// TwinCAT 3 PLC project PidTests
// ProgramVersion: 3.1.4026.22
// libraries:
//   Tc2_Standard, * (Beckhoff Automation GmbH)
//   Tc2_System, * (Beckhoff Automation GmbH)
//   TcUnit, * (www.tcunit.org)
//   T2Pid_Plc,newest,Tc3 Project
// project tree:
//   / PlcTask.TcTTO
//   POUs/ FB_PidTests.TcPOU, MAIN.TcPOU
// real-time tasks:
//   TASK PlcTask: cycle T#10ms, priority 20, ADS port 350

CONFIGURATION PidTests
    RESOURCE PLC ON TwinCAT3
        TASK PlcTask(INTERVAL := T#10ms, PRIORITY := 20);
        PROGRAM MAIN WITH PlcTask : MAIN;
    END_RESOURCE
END_CONFIGURATION

// ---- POUs/MAIN.TcPOU
PROGRAM MAIN
VAR
    suite : FB_PidTests;
END_VAR

suite();
TcUnit.RUN();

END_PROGRAM

// ---- POUs/FB_PidTests.TcPOU
FUNCTION_BLOCK FB_PidTests EXTENDS TcUnit.FB_TestSuite
VAR
    pid       : T2Pid_Plc.FB_Pid;
    iPid      : T2Pid_Plc.I_Pid;
    output    : LREAL;
    output2   : LREAL;
    integral  : LREAL;
    saturated : BOOL;
    i         : DINT;
END_VAR

PProportionalOnly();
OutputClampsToMax();
OutputClampsToMin();
IntegralAccumulates();
AntiWindupHoldsIntegral();
DerivativeOnMeasurementNoSetpointSpike();
ReverseModeFlipsSign();
ResetClearsIntegral();
SetterRejectsNegativeKp();
IsSaturatedReflectsClampState();
CyclicReachableThroughInterface();

METHOD AntiWindupHoldsIntegral : BOOL
VAR
    integral : LREAL;
    i : DINT;
END_VAR
IF TEST_ORDERED(__POUNAME()) THEN
    pid.Reset();
    pid.Kp := 0.0;
    pid.Ki := 10.0;
    pid.Kd := 0.0;
    pid.Mode := 0;
    pid.OutputMin := -1.0;
    pid.OutputMax := 1.0;
    // Drive into saturation: with Ki=10 and error=1, a single 0.1s tick
    // would produce output 1.0 (at clamp). Twenty more ticks should
    // not grow the integral once saturated.
    FOR i := 1 TO 20 DO
        pid.Update(setpoint := 1.0, measurement := 0.0, deltaT := 0.1);
    END_FOR
    integral := pid.IntegralTerm;
    AssertTrue(Condition := integral <= 0.2,
        Message := 'Anti-windup should hold integral at/near saturation point, not let it grow');
    TEST_FINISHED();
END_IF
END_METHOD

METHOD CyclicReachableThroughInterface : BOOL
VAR
    direct    : LREAL;
    viaIface  : LREAL;
END_VAR
IF TEST_ORDERED(__POUNAME()) THEN
    pid.Reset();
    pid.Kp := 3.0;
    pid.Ki := 0.0;
    pid.Kd := 0.0;
    pid.Mode := 0;
    pid.OutputMin := -100.0;
    pid.OutputMax := 100.0;
    direct := pid.Update(setpoint := 1.0, measurement := 0.0, deltaT := 0.1);

    pid.Reset();
    iPid := pid;  // FB_Pid IMPLEMENTS I_Pid required
    viaIface := iPid.Update(setpoint := 1.0, measurement := 0.0, deltaT := 0.1);

    AssertEquals_LREAL(Expected := direct, Actual := viaIface, Delta := 1E-9,
        Message := 'Same Update inputs through pid and iPid must give the same output');
    TEST_FINISHED();
END_IF
END_METHOD

METHOD DerivativeOnMeasurementNoSetpointSpike : BOOL
VAR
    output : LREAL;
    output2 : LREAL;
END_VAR
IF TEST_ORDERED(__POUNAME()) THEN
    pid.Reset();
    pid.Kp := 0.0;
    pid.Ki := 0.0;
    pid.Kd := 1.0;
    pid.Mode := 0;
    pid.OutputMin := -100.0;
    pid.OutputMax := 100.0;
    // Steady state: setpoint=0, measurement=0.
    pid.Update(setpoint := 0.0, measurement := 0.0, deltaT := 0.1);
    // Step the SETPOINT. With derivative-on-error this would produce
    // a large spike (d_error/dt ~ 100). With derivative-on-measurement
    // the derivative is computed from -dMeasurement/dt, which is 0.
    output := pid.Update(setpoint := 10.0, measurement := 0.0, deltaT := 0.1);
    AssertTrue(Condition := ABS(output) < 1.0,
        Message := 'Derivative-on-measurement: setpoint step must NOT cause D-kick');
    TEST_FINISHED();
END_IF
END_METHOD

METHOD IntegralAccumulates : BOOL
VAR
    integral : LREAL;
    i : DINT;
END_VAR
IF TEST_ORDERED(__POUNAME()) THEN
    pid.Reset();
    pid.Kp := 0.0;
    pid.Ki := 1.0;
    pid.Kd := 0.0;
    pid.Mode := 0;
    pid.OutputMin := -100.0;
    pid.OutputMax := 100.0;
    FOR i := 1 TO 10 DO
        pid.Update(setpoint := 1.0, measurement := 0.0, deltaT := 0.1);
    END_FOR
    integral := pid.IntegralTerm;
    AssertEquals_LREAL(Expected := 1.0, Actual := integral, Delta := 0.05,
        Message := 'I-only Ki=1 error=1 for 10x0.1s should integrate to ~1.0');
    TEST_FINISHED();
END_IF
END_METHOD

METHOD IsSaturatedReflectsClampState : BOOL
VAR
    saturated : BOOL;
END_VAR
IF TEST_ORDERED(__POUNAME()) THEN
    pid.Reset();
    pid.Kp := 1.0;
    pid.Ki := 0.0;
    pid.Kd := 0.0;
    pid.Mode := 0;
    pid.OutputMin := -10.0;
    pid.OutputMax := 10.0;
    // Small error, output well within limits.
    pid.Update(setpoint := 1.0, measurement := 0.0, deltaT := 0.1);
    saturated := pid.IsSaturated;
    AssertFalse(Condition := saturated,
        Message := 'IsSaturated should be FALSE when output is within OutputMin..OutputMax');
    // Now saturate the output.
    pid.Update(setpoint := 100.0, measurement := 0.0, deltaT := 0.1);
    saturated := pid.IsSaturated;
    AssertTrue(Condition := saturated,
        Message := 'IsSaturated should be TRUE once the output is clamped to OutputMax');
    TEST_FINISHED();
END_IF
END_METHOD

METHOD OutputClampsToMax : BOOL
VAR
    output : LREAL;
END_VAR
IF TEST_ORDERED(__POUNAME()) THEN
    pid.Reset();
    pid.Kp := 2.0;
    pid.Ki := 0.0;
    pid.Kd := 0.0;
    pid.Mode := 0;
    pid.OutputMin := -5.0;
    pid.OutputMax := 5.0;
    output := pid.Update(setpoint := 100.0, measurement := 0.0, deltaT := 0.1);
    AssertEquals_LREAL(Expected := 5.0, Actual := output, Delta := 1E-6,
        Message := 'Output should clamp to OutputMax on large positive error');
    TEST_FINISHED();
END_IF
END_METHOD

METHOD OutputClampsToMin : BOOL
VAR
    output : LREAL;
END_VAR
IF TEST_ORDERED(__POUNAME()) THEN
    pid.Reset();
    pid.Kp := 2.0;
    pid.Ki := 0.0;
    pid.Kd := 0.0;
    pid.Mode := 0;
    pid.OutputMin := -5.0;
    pid.OutputMax := 5.0;
    output := pid.Update(setpoint := -100.0, measurement := 0.0, deltaT := 0.1);
    AssertEquals_LREAL(Expected := -5.0, Actual := output, Delta := 1E-6,
        Message := 'Output should clamp to OutputMin on large negative error');
    TEST_FINISHED();
END_IF
END_METHOD

METHOD PProportionalOnly : BOOL
VAR
    output : LREAL;
END_VAR
IF TEST_ORDERED(__POUNAME()) THEN
    pid.Reset();
    pid.Kp := 2.0;
    pid.Ki := 0.0;
    pid.Kd := 0.0;
    pid.Mode := 0;
    pid.OutputMin := -100.0;
    pid.OutputMax := 100.0;
    output := pid.Update(setpoint := 1.0, measurement := 0.0, deltaT := 0.1);
    AssertEquals_LREAL(Expected := 2.0, Actual := output, Delta := 1E-6,
        Message := 'P-only Kp=2 error=1 should yield output=2');
    TEST_FINISHED();
END_IF
END_METHOD

METHOD ResetClearsIntegral : BOOL
VAR
    integral : LREAL;
    i : DINT;
END_VAR
IF TEST_ORDERED(__POUNAME()) THEN
    pid.Kp := 0.0;
    pid.Ki := 1.0;
    pid.Kd := 0.0;
    pid.Mode := 0;
    pid.OutputMin := -100.0;
    pid.OutputMax := 100.0;
    FOR i := 1 TO 5 DO
        pid.Update(setpoint := 1.0, measurement := 0.0, deltaT := 0.1);
    END_FOR
    AssertTrue(Condition := pid.IntegralTerm > 0.0,
        Message := 'Integral must be non-zero before Reset for this test to be meaningful');
    pid.Reset();
    integral := pid.IntegralTerm;
    AssertEquals_LREAL(Expected := 0.0, Actual := integral, Delta := 1E-9,
        Message := 'Reset must zero the integral term');
    TEST_FINISHED();
END_IF
END_METHOD

METHOD ReverseModeFlipsSign : BOOL
VAR
    output : LREAL;
END_VAR
IF TEST_ORDERED(__POUNAME()) THEN
    pid.Reset();
    pid.Kp := 2.0;
    pid.Ki := 0.0;
    pid.Kd := 0.0;
    pid.Mode := 1;  // reverse
    pid.OutputMin := -100.0;
    pid.OutputMax := 100.0;
    output := pid.Update(setpoint := 1.0, measurement := 0.0, deltaT := 0.1);
    AssertEquals_LREAL(Expected := -2.0, Actual := output, Delta := 1E-6,
        Message := 'Reverse mode should flip the sign of the controller output');
    TEST_FINISHED();
END_IF
END_METHOD

METHOD SetterRejectsNegativeKp : BOOL
IF TEST_ORDERED(__POUNAME()) THEN
    pid.Kp := 0.5;
    pid.Kp := -1.0;  // setter must reject this
    AssertEquals_LREAL(Expected := 0.5, Actual := pid.Kp, Delta := 1E-9,
        Message := 'Setter must reject negative Kp; existing value preserved');
    TEST_FINISHED();
END_IF
END_METHOD

END_FUNCTION_BLOCK
